FUNCTION_BLOCK ABSTRACT CoE_property IMPLEMENTS I_CoE_property
VAR_INPUT
END_VAR
VAR_OUTPUT
END_VAR
VAR
	_SubIndex 		: BYTE;
	_Index			: WORD;
	_init_done		: BOOL;
	_neg_replay		: f_trig;
	_SlaveAddress	: WORD;
	_propertyType	: UINT;
	_pollingInterval: TIME;
	_I_CoE_communication_handler: I_CoE_communication_handler;
	
	_read_errId		: UDINT;
	_write_errId	: UDINT;
	_init_state		: INT;
	
	_valueToWrite 	: CoE_buffer_type_cast_union;

	pollingTimer: ton;
	
	errId: INT;
END_VAR

CASE _propertyType OF 
	0:  // cashed 
		;
	
	1:  // polling 
		pollingTimer(IN:=NOT pollingTimer.q, PT:=_pollingInterval);
		IF pollingTimer.Q THEN
			IF THIS^._I_CoE_communication_handler <> 0 THEN 
				THIS^._I_CoE_communication_handler.add_read_request(THIS^);
			ELSE
				errId:=1;
			END_IF
		END_IF
	
	2: // on request
		IF THIS^._I_CoE_communication_handler <> 0 THEN 
			THIS^._I_CoE_communication_handler.add_read_request(THIS^);
		ELSE
			errId:=1; 
		END_IF

ELSE
	errId:=2; 
END_CASE

PROPERTY CoE_communication_handler : I_CoE_communication_handler
GET
CoE_communication_handler:=_I_CoE_communication_handler;
END_GET
SET
_I_CoE_communication_handler:=CoE_communication_handler;
END_SET
END_PROPERTY

PROPERTY dataTypeSize : UINT
GET
END_GET
END_PROPERTY

METHOD FB_init : BOOL
VAR_INPUT
	bInitRetains 			: BOOL; // if TRUE, the retain variables are initialized (warm start / cold start)
	bInCopyCode 			: BOOL;  // if TRUE, the instance afterwards gets moved into the copy code (online change)
	Index					: WORD;
	SubIndex				: BYTE;
	writable				: BOOL;
	propertyType			: UINT;
	pollingInterval 		: TIME;
END_VAR
_Index:=Index;
_SubIndex:=SubIndex;
_propertyType:=propertyType;
_pollingInterval:=pollingInterval;
END_METHOD

METHOD handle_read_callback : BOOL
VAR_INPUT
	pt_buffer : POINTER TO CoE_buffer_type_cast_union;
	errId : UDINT;
END_VAR
END_METHOD

METHOD handle_write_callback : BOOL
VAR_INPUT
	errId	: UDINT;
END_VAR
_write_errId:=errId;
END_METHOD

PROPERTY Index : word
GET
Index:=_Index;
END_GET
SET
_Index:=Index;
END_SET
END_PROPERTY

PROPERTY init_done : BOOL
GET
init_done := _init_done;
END_GET
END_PROPERTY

METHOD reinit : BOOL
VAR_OUTPUT
	errId: UDINT;
END_VAR

CASE _init_state OF 
	0:  // add read request and continue
		_init_done:=FALSE;
		reinit:=FALSE;
		IF THIS^._I_CoE_communication_handler <> 0 THEN 
			THIS^._I_CoE_communication_handler.add_read_request(THIS^);
		ELSE
			errId:=1;
		END_IF
		_init_state := 10;
		
	10: // wait for read callback
		reinit:=TRUE;
		errId:=_read_errId;
		_init_state := 0;
END_CASE
END_METHOD

METHOD run : BOOL
THIS^();
END_METHOD

PROPERTY SlaveAddress : uint
GET
SlaveAddress:=_SlaveAddress;
END_GET
SET
_SlaveAddress:=SlaveAddress;
END_SET
END_PROPERTY

PROPERTY SubIndex : BYTE
GET
SubIndex:=_SubIndex;
END_GET
SET
_SubIndex:=SubIndex;
END_SET
END_PROPERTY

PROPERTY valueToWrite : CoE_buffer_type_cast_union
GET
valueToWrite := _valueToWrite;
END_GET
END_PROPERTY

END_FUNCTION_BLOCK

(* stored: Version 1.1.0.1, ProductVersion 3.1.4024.6
   POU CoE_property: Id {7290e4d7-edb9-0644-02c0-672d2dd6d3bf}, SpecialFunc None
   Property CoE_communication_handler: Id {41443338-f88e-057f-2a53-60a637a72aec}
   Get Get: Id {f1d614f3-ef34-0c15-379c-8bb05239b83a}
   Set Set: Id {2a291f26-afc4-0090-3fb7-9dbae000bc11}
   Property dataTypeSize: Id {c8c62b6f-a562-0288-24b7-a97cdf714276}
   Get Get: Id {82523ad0-d4b6-0490-05f6-e1f39508487e}
   Method FB_init: Id {a3c72071-8363-0c5f-2ef3-dfe5d0b2b01a}
   Method handle_read_callback: Id {358e0672-e92e-0990-3d90-6a809c7ca1fb}
   Method handle_write_callback: Id {f74faa57-7cc3-0d8b-3ecc-005cac59e305}
   Property Index: Id {6009d123-ed20-0cfb-2d9f-975880c33335}
   Get Get: Id {93e74eed-a441-0466-3ff2-acca7aa2f70f}
   Set Set: Id {b0390769-4a06-0c12-0992-4445a0964b07}
   Property init_done: Id {2272e174-b6d6-026b-1bd7-e6f0499f6eab}
   Get Get: Id {b00b0881-afce-0686-1dee-90c84869b238}
   Method reinit: Id {30436167-4235-0089-245f-f4e6c137a925}
   Method run: Id {6d816fe4-c312-0232-0c99-9a2e3f2db29f}
   Property SlaveAddress: Id {c15f8ec3-c06d-090d-2a91-e412f7c9f477}
   Get Get: Id {4709cc48-424c-0841-2c5c-d0657830a023}
   Set Set: Id {d4171903-85fd-03fd-120b-0b1b46a254cf}
   Property SubIndex: Id {a962e5da-e69b-0444-170f-71416eb83565}
   Get Get: Id {4a058a33-93ff-02af-3339-83d7fe3bdce4}
   Set Set: Id {171b2b00-46fd-07f1-3589-e75c1ffb6e3a}
   Property valueToWrite: Id {f671e68f-34dc-08aa-3fa7-0dbc6c977bb5}
   Get Get: Id {dae09c31-b983-0ff6-240f-1eb3ae3a0c98} *)
